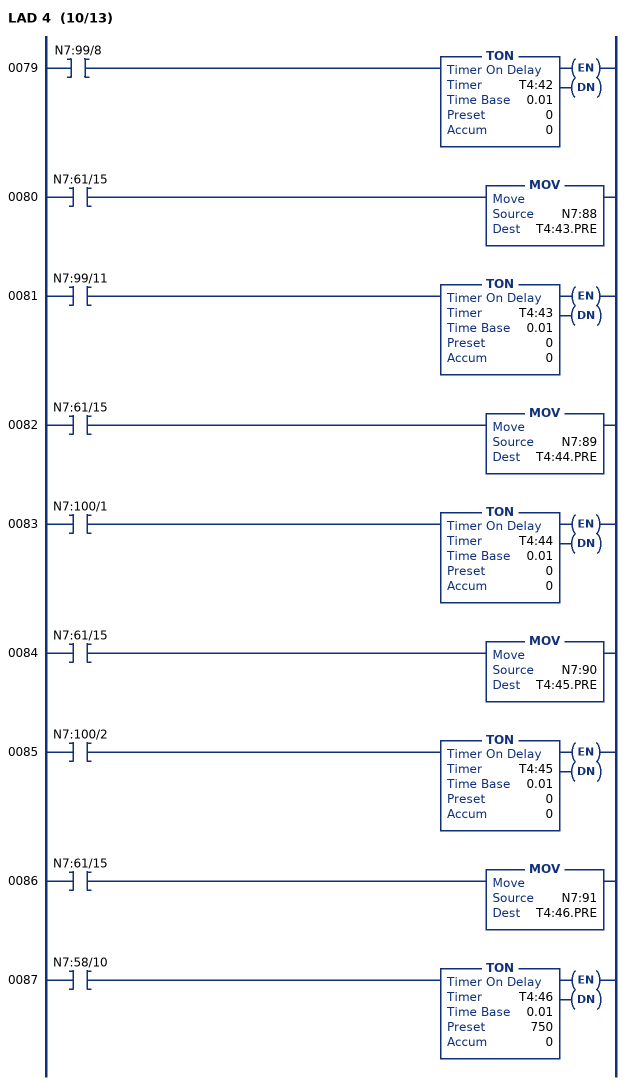
% Rung: 79 %
SOR XIC N7:99/8 TON T4:42 0.01 0 0 EOR
% Rung: 80 %
SOR XIC N7:61/15 MOV N7:88 T4:43.PRE EOR
% Rung: 81 %
SOR XIC N7:99/11 TON T4:43 0.01 0 0 EOR
% Rung: 82 %
SOR XIC N7:61/15 MOV N7:89 T4:44.PRE EOR
% Rung: 83 %
SOR XIC N7:100/1 TON T4:44 0.01 0 0 EOR
% Rung: 84 %
SOR XIC N7:61/15 MOV N7:90 T4:45.PRE EOR
% Rung: 85 %
SOR XIC N7:100/2 TON T4:45 0.01 0 0 EOR
% Rung: 86 %
SOR XIC N7:61/15 MOV N7:91 T4:46.PRE EOR
% Rung: 87 %
SOR XIC N7:58/10 TON T4:46 0.01 750 0 EOR

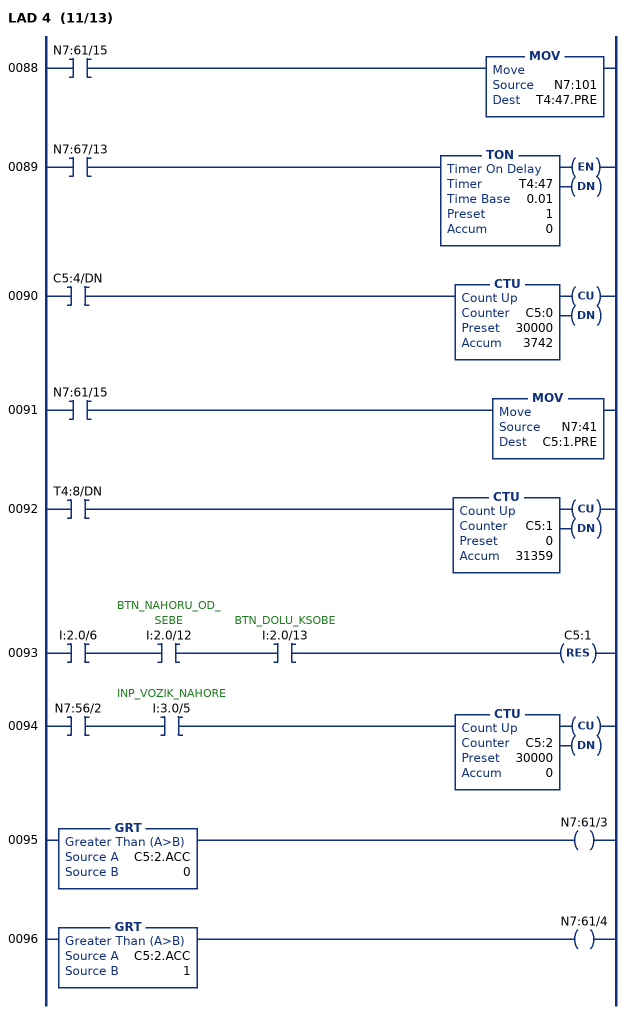
% Rung: 88 %
SOR XIC N7:61/15 MOV N7:101 T4:47.PRE EOR
% Rung: 89 %
SOR XIC N7:67/13 TON T4:47 0.01 1 0 EOR
% Rung: 90 %
SOR XIC C5:4/DN CTU C5:0 30000 3742 EOR
% Rung: 91 %
SOR XIC N7:61/15 MOV N7:41 C5:1.PRE EOR
% Rung: 92 %
SOR XIC T4:8/DN CTU C5:1 0 31359 EOR
% Rung: 93 %
SOR XIC I:2.0/6 XIC I:2.0/12 XIC I:2.0/13 RES C5:1 EOR
%   I:2.0/12  BTN_NAHORU_OD_SEBE %
%   I:2.0/13  BTN_DOLU_KSOBE %
% Rung: 94 %
SOR XIC N7:56/2 XIC I:3.0/5 CTU C5:2 30000 0 EOR
%   I:3.0/5  INP_VOZIK_NAHORE %
% Rung: 95 %
SOR GRT C5:2.ACC 0 OTE N7:61/3 EOR
% Rung: 96 %
SOR GRT C5:2.ACC 1 OTE N7:61/4 EOR

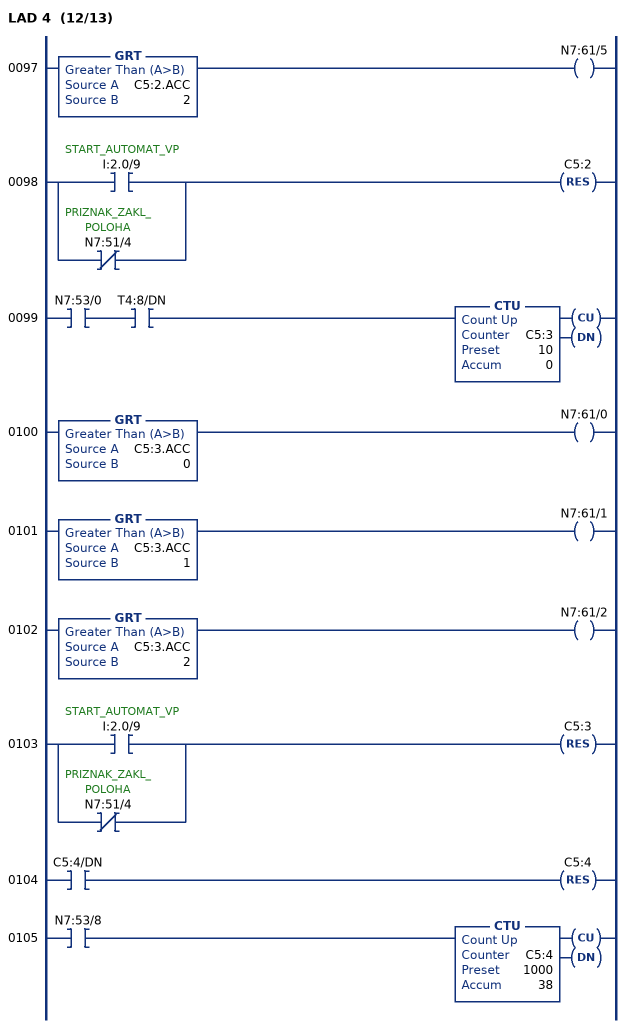
% Rung: 97 %
SOR GRT C5:2.ACC 2 OTE N7:61/5 EOR
% Rung: 98 %
SOR BST XIC I:2.0/9 NXB XIO N7:51/4 BND RES C5:2 EOR
%   I:2.0/9  START_AUTOMAT_VP %
%   N7:51/4  PRIZNAK_ZAKL_POLOHA %
% Rung: 99 %
SOR XIC N7:53/0 XIC T4:8/DN CTU C5:3 10 0 EOR
% Rung: 100 %
SOR GRT C5:3.ACC 0 OTE N7:61/0 EOR
% Rung: 101 %
SOR GRT C5:3.ACC 1 OTE N7:61/1 EOR
% Rung: 102 %
SOR GRT C5:3.ACC 2 OTE N7:61/2 EOR
% Rung: 103 %
SOR BST XIC I:2.0/9 NXB XIO N7:51/4 BND RES C5:3 EOR
%   I:2.0/9  START_AUTOMAT_VP %
%   N7:51/4  PRIZNAK_ZAKL_POLOHA %
% Rung: 104 %
SOR XIC C5:4/DN RES C5:4 EOR
% Rung: 105 %
SOR XIC N7:53/8 CTU C5:4 1000 38 EOR

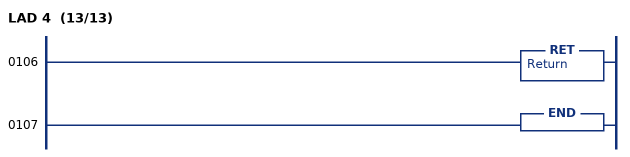
% Rung: 106 %
SOR RET EOR
% Rung: 107 %
SOR END EOR

LADDER 5
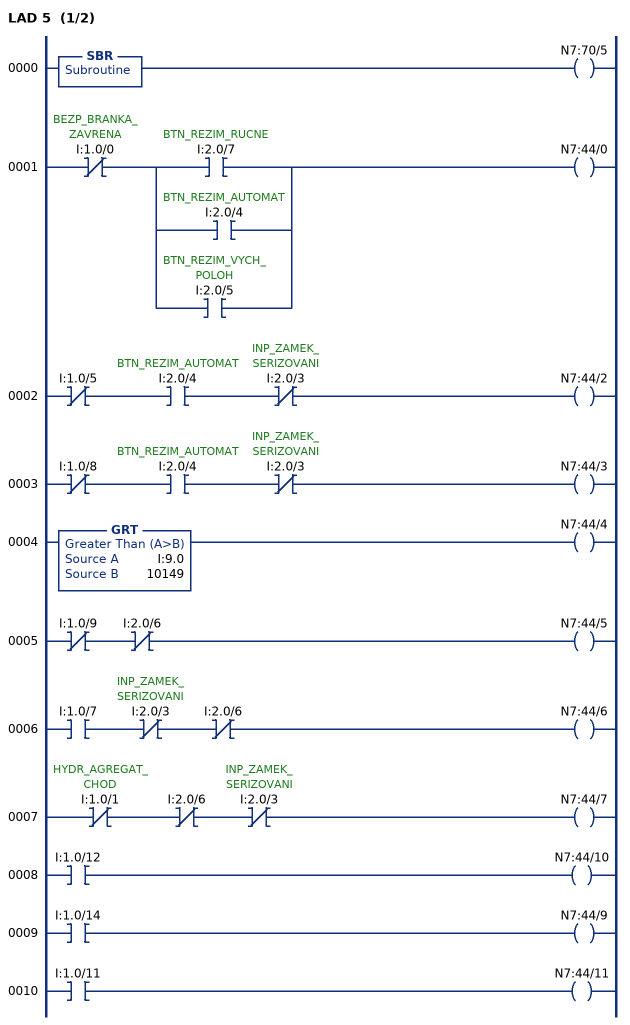
% Rung: 0 %
SOR SBR OTE N7:70/5 EOR
% Rung: 1 %
SOR XIO I:1.0/0 BST XIC I:2.0/7 NXB XIC I:2.0/4 NXB XIC I:2.0/5 BND OTE N7:44/0 EOR
%   I:1.0/0  BEZP_BRANKA_ZAVRENA %
%   I:2.0/7  BTN_REZIM_RUCNE %
%   I:2.0/4  BTN_REZIM_AUTOMAT %
%   I:2.0/5  BTN_REZIM_VYCH_POLOH %
% Rung: 2 %
SOR XIO I:1.0/5 XIC I:2.0/4 XIO I:2.0/3 OTE N7:44/2 EOR
%   I:2.0/4  BTN_REZIM_AUTOMAT %
%   I:2.0/3  INP_ZAMEK_SERIZOVANI %
% Rung: 3 %
SOR XIO I:1.0/8 XIC I:2.0/4 XIO I:2.0/3 OTE N7:44/3 EOR
%   I:2.0/4  BTN_REZIM_AUTOMAT %
%   I:2.0/3  INP_ZAMEK_SERIZOVANI %
% Rung: 4 %
SOR GRT I:9.0 10149 OTE N7:44/4 EOR
% Rung: 5 %
SOR XIO I:1.0/9 XIO I:2.0/6 OTE N7:44/5 EOR
% Rung: 6 %
SOR XIC I:1.0/7 XIO I:2.0/3 XIO I:2.0/6 OTE N7:44/6 EOR
%   I:2.0/3  INP_ZAMEK_SERIZOVANI %
% Rung: 7 %
SOR XIO I:1.0/1 XIO I:2.0/6 XIO I:2.0/3 OTE N7:44/7 EOR
%   I:1.0/1  HYDR_AGREGAT_CHOD %
%   I:2.0/3  INP_ZAMEK_SERIZOVANI %
% Rung: 8 %
SOR XIC I:1.0/12 OTE N7:44/10 EOR
% Rung: 9 %
SOR XIC I:1.0/14 OTE N7:44/9 EOR
% Rung: 10 %
SOR XIC I:1.0/11 OTE N7:44/11 EOR

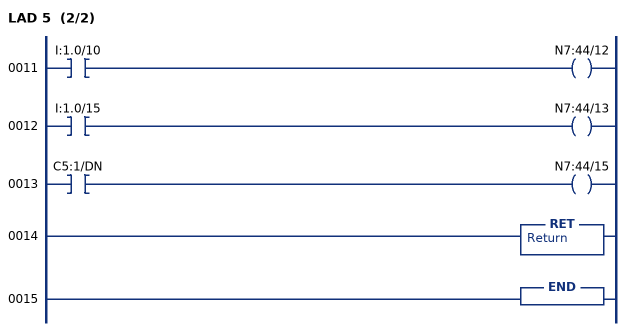
% Rung: 11 %
SOR XIC I:1.0/10 OTE N7:44/12 EOR
% Rung: 12 %
SOR XIC I:1.0/15 OTE N7:44/13 EOR
% Rung: 13 %
SOR XIC C5:1/DN OTE N7:44/15 EOR
% Rung: 14 %
SOR RET EOR
% Rung: 15 %
SOR END EOR

LADDER 6
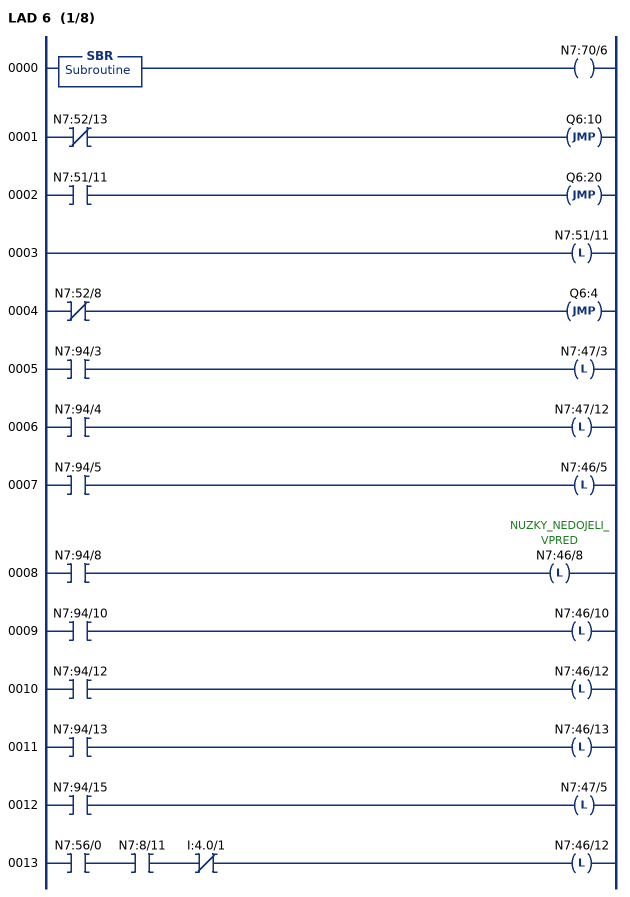
% Rung: 0 %
SOR SBR OTE N7:70/6 EOR
% Rung: 1 %
SOR XIO N7:52/13 JMP Q6:10 EOR
% Rung: 2 %
SOR XIC N7:51/11 JMP Q6:20 EOR
% Rung: 3 %
SOR OTL N7:51/11 EOR
% Rung: 4 %
SOR XIO N7:52/8 JMP Q6:4 EOR
% Rung: 5 %
SOR XIC N7:94/3 OTL N7:47/3 EOR
% Rung: 6 %
SOR XIC N7:94/4 OTL N7:47/12 EOR
% Rung: 7 %
SOR XIC N7:94/5 OTL N7:46/5 EOR
% Rung: 8 %
SOR XIC N7:94/8 OTL N7:46/8 EOR
%   N7:46/8  NUZKY_NEDOJELI_VPRED %
% Rung: 9 %
SOR XIC N7:94/10 OTL N7:46/10 EOR
% Rung: 10 %
SOR XIC N7:94/12 OTL N7:46/12 EOR
% Rung: 11 %
SOR XIC N7:94/13 OTL N7:46/13 EOR
% Rung: 12 %
SOR XIC N7:94/15 OTL N7:47/5 EOR
% Rung: 13 %
SOR XIC N7:56/0 XIC N7:8/11 XIO I:4.0/1 OTL N7:46/12 EOR

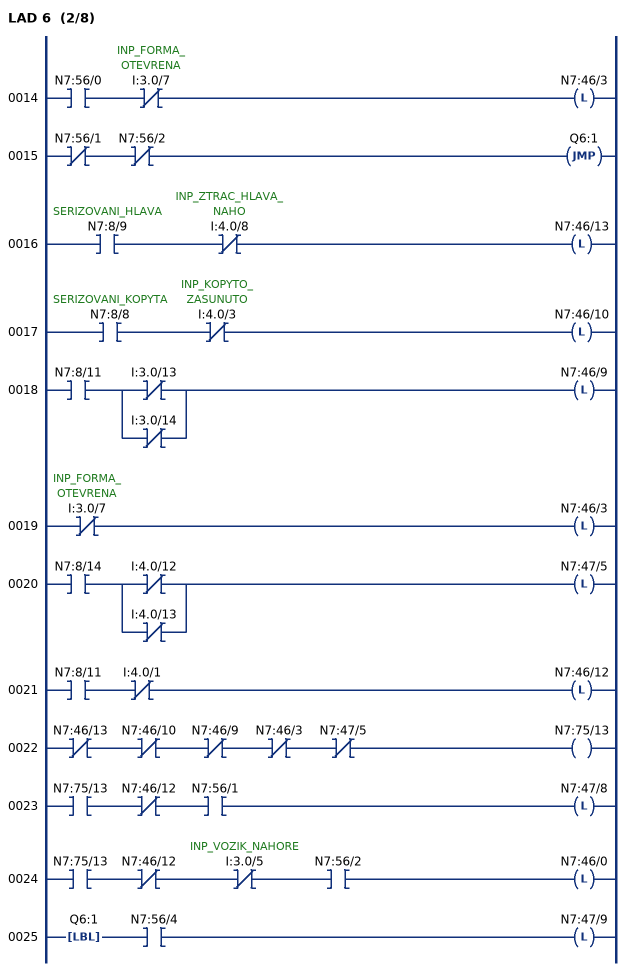
% Rung: 14 %
SOR XIC N7:56/0 XIO I:3.0/7 OTL N7:46/3 EOR
%   I:3.0/7  INP_FORMA_OTEVRENA %
% Rung: 15 %
SOR XIO N7:56/1 XIO N7:56/2 JMP Q6:1 EOR
% Rung: 16 %
SOR XIC N7:8/9 XIO I:4.0/8 OTL N7:46/13 EOR
%   N7:8/9  SERIZOVANI_HLAVA %
%   I:4.0/8  INP_ZTRAC_HLAVA_NAHO %
% Rung: 17 %
SOR XIC N7:8/8 XIO I:4.0/3 OTL N7:46/10 EOR
%   N7:8/8  SERIZOVANI_KOPYTA %
%   I:4.0/3  INP_KOPYTO_ZASUNUTO %
% Rung: 18 %
SOR XIC N7:8/11 BST XIO I:3.0/13 NXB XIO I:3.0/14 BND OTL N7:46/9 EOR
% Rung: 19 %
SOR XIO I:3.0/7 OTL N7:46/3 EOR
%   I:3.0/7  INP_FORMA_OTEVRENA %
% Rung: 20 %
SOR XIC N7:8/14 BST XIO I:4.0/12 NXB XIO I:4.0/13 BND OTL N7:47/5 EOR
% Rung: 21 %
SOR XIC N7:8/11 XIO I:4.0/1 OTL N7:46/12 EOR
% Rung: 22 %
SOR XIO N7:46/13 XIO N7:46/10 XIO N7:46/9 XIO N7:46/3 XIO N7:47/5 OTE N7:75/13 EOR
% Rung: 23 %
SOR XIC N7:75/13 XIO N7:46/12 XIC N7:56/1 OTL N7:47/8 EOR
% Rung: 24 %
SOR XIC N7:75/13 XIO N7:46/12 XIO I:3.0/5 XIC N7:56/2 OTL N7:46/0 EOR
%   I:3.0/5  INP_VOZIK_NAHORE %
% Rung: 25 %
SOR LBL Q6:1 XIC N7:56/4 OTL N7:47/9 EOR

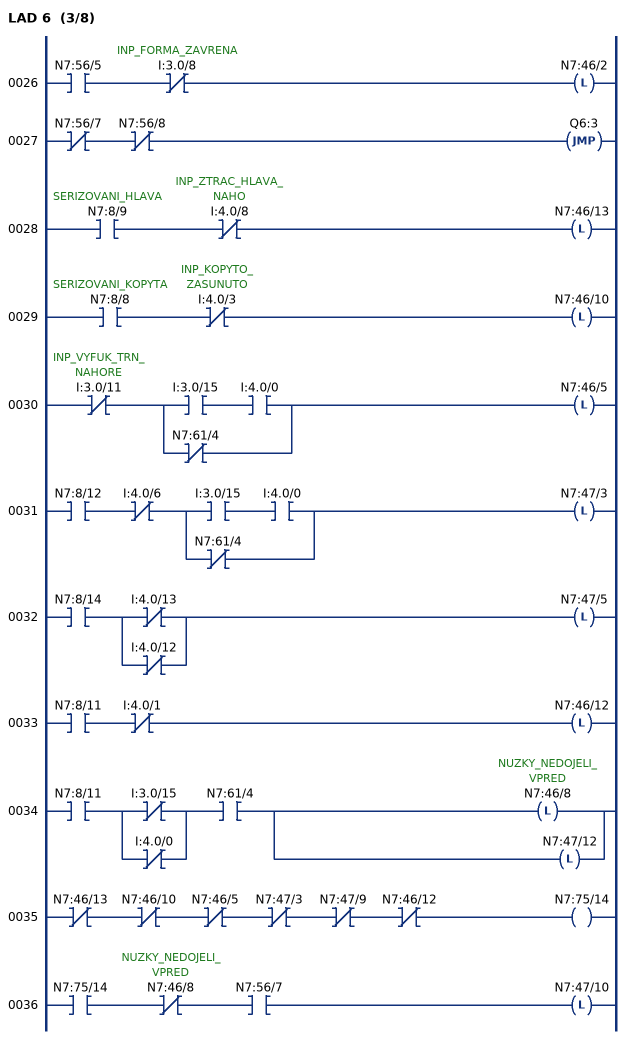
% Rung: 26 %
SOR XIC N7:56/5 XIO I:3.0/8 OTL N7:46/2 EOR
%   I:3.0/8  INP_FORMA_ZAVRENA %
% Rung: 27 %
SOR XIO N7:56/7 XIO N7:56/8 JMP Q6:3 EOR
% Rung: 28 %
SOR XIC N7:8/9 XIO I:4.0/8 OTL N7:46/13 EOR
%   N7:8/9  SERIZOVANI_HLAVA %
%   I:4.0/8  INP_ZTRAC_HLAVA_NAHO %
% Rung: 29 %
SOR XIC N7:8/8 XIO I:4.0/3 OTL N7:46/10 EOR
%   N7:8/8  SERIZOVANI_KOPYTA %
%   I:4.0/3  INP_KOPYTO_ZASUNUTO %
% Rung: 30 %
SOR XIO I:3.0/11 BST XIC I:3.0/15 XIC I:4.0/0 NXB XIO N7:61/4 BND OTL N7:46/5 EOR
%   I:3.0/11  INP_VYFUK_TRN_NAHORE %
% Rung: 31 %
SOR XIC N7:8/12 XIO I:4.0/6 BST XIC I:3.0/15 XIC I:4.0/0 NXB XIO N7:61/4 BND OTL N7:47/3 EOR
% Rung: 32 %
SOR XIC N7:8/14 BST XIO I:4.0/13 NXB XIO I:4.0/12 BND OTL N7:47/5 EOR
% Rung: 33 %
SOR XIC N7:8/11 XIO I:4.0/1 OTL N7:46/12 EOR
% Rung: 34 %
SOR XIC N7:8/11 BST XIO I:3.0/15 NXB XIO I:4.0/0 BND XIC N7:61/4 BST OTL N7:46/8 NXB OTL N7:47/12 BND EOR
%   N7:46/8  NUZKY_NEDOJELI_VPRED %
% Rung: 35 %
SOR XIO N7:46/13 XIO N7:46/10 XIO N7:46/5 XIO N7:47/3 XIO N7:47/9 XIO N7:46/12 OTE N7:75/14 EOR
% Rung: 36 %
SOR XIC N7:75/14 XIO N7:46/8 XIC N7:56/7 OTL N7:47/10 EOR
%   N7:46/8  NUZKY_NEDOJELI_VPRED %

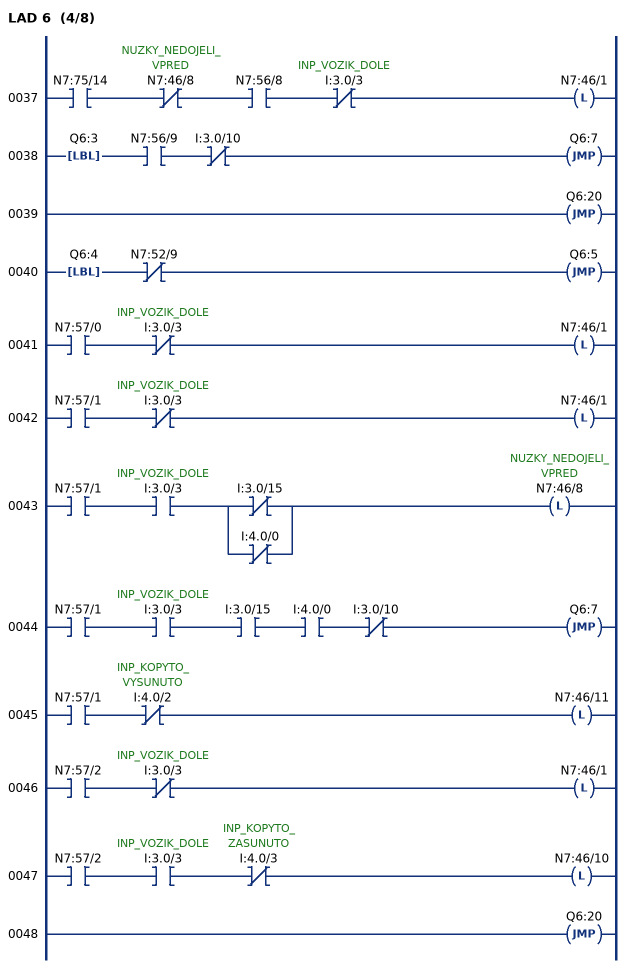
% Rung: 37 %
SOR XIC N7:75/14 XIO N7:46/8 XIC N7:56/8 XIO I:3.0/3 OTL N7:46/1 EOR
%   N7:46/8  NUZKY_NEDOJELI_VPRED %
%   I:3.0/3  INP_VOZIK_DOLE %
% Rung: 38 %
SOR LBL Q6:3 XIC N7:56/9 XIO I:3.0/10 JMP Q6:7 EOR
% Rung: 39 %
SOR JMP Q6:20 EOR
% Rung: 40 %
SOR LBL Q6:4 XIO N7:52/9 JMP Q6:5 EOR
% Rung: 41 %
SOR XIC N7:57/0 XIO I:3.0/3 OTL N7:46/1 EOR
%   I:3.0/3  INP_VOZIK_DOLE %
% Rung: 42 %
SOR XIC N7:57/1 XIO I:3.0/3 OTL N7:46/1 EOR
%   I:3.0/3  INP_VOZIK_DOLE %
% Rung: 43 %
SOR XIC N7:57/1 XIC I:3.0/3 BST XIO I:3.0/15 NXB XIO I:4.0/0 BND OTL N7:46/8 EOR
%   I:3.0/3  INP_VOZIK_DOLE %
%   N7:46/8  NUZKY_NEDOJELI_VPRED %
% Rung: 44 %
SOR XIC N7:57/1 XIC I:3.0/3 XIC I:3.0/15 XIC I:4.0/0 XIO I:3.0/10 JMP Q6:7 EOR
%   I:3.0/3  INP_VOZIK_DOLE %
% Rung: 45 %
SOR XIC N7:57/1 XIO I:4.0/2 OTL N7:46/11 EOR
%   I:4.0/2  INP_KOPYTO_VYSUNUTO %
% Rung: 46 %
SOR XIC N7:57/2 XIO I:3.0/3 OTL N7:46/1 EOR
%   I:3.0/3  INP_VOZIK_DOLE %
% Rung: 47 %
SOR XIC N7:57/2 XIC I:3.0/3 XIO I:4.0/3 OTL N7:46/10 EOR
%   I:3.0/3  INP_VOZIK_DOLE %
%   I:4.0/3  INP_KOPYTO_ZASUNUTO %
% Rung: 48 %
SOR JMP Q6:20 EOR

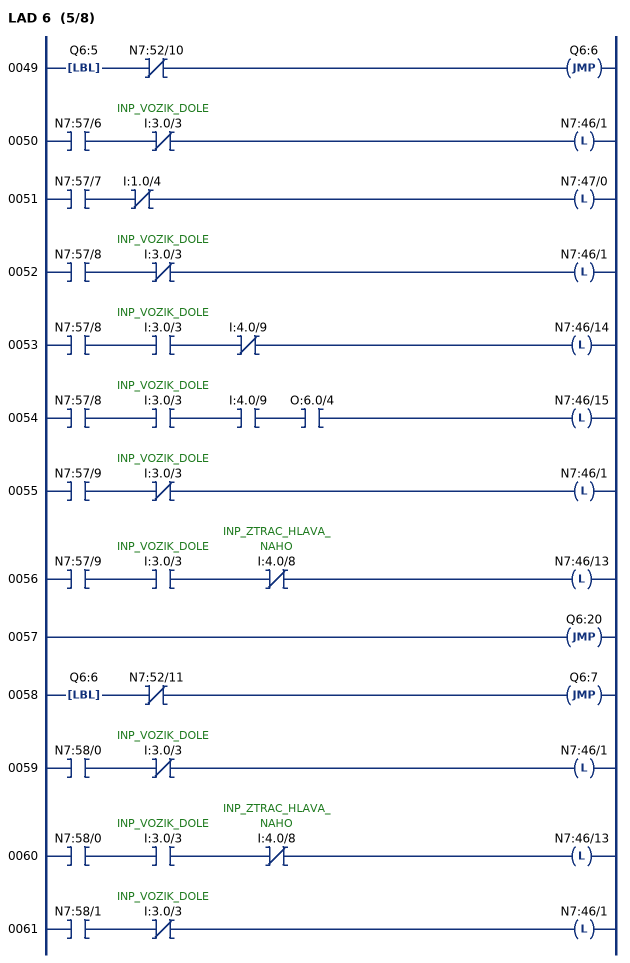
% Rung: 49 %
SOR LBL Q6:5 XIO N7:52/10 JMP Q6:6 EOR
% Rung: 50 %
SOR XIC N7:57/6 XIO I:3.0/3 OTL N7:46/1 EOR
%   I:3.0/3  INP_VOZIK_DOLE %
% Rung: 51 %
SOR XIC N7:57/7 XIO I:1.0/4 OTL N7:47/0 EOR
% Rung: 52 %
SOR XIC N7:57/8 XIO I:3.0/3 OTL N7:46/1 EOR
%   I:3.0/3  INP_VOZIK_DOLE %
% Rung: 53 %
SOR XIC N7:57/8 XIC I:3.0/3 XIO I:4.0/9 OTL N7:46/14 EOR
%   I:3.0/3  INP_VOZIK_DOLE %
% Rung: 54 %
SOR XIC N7:57/8 XIC I:3.0/3 XIC I:4.0/9 XIC O:6.0/4 OTL N7:46/15 EOR
%   I:3.0/3  INP_VOZIK_DOLE %
% Rung: 55 %
SOR XIC N7:57/9 XIO I:3.0/3 OTL N7:46/1 EOR
%   I:3.0/3  INP_VOZIK_DOLE %
% Rung: 56 %
SOR XIC N7:57/9 XIC I:3.0/3 XIO I:4.0/8 OTL N7:46/13 EOR
%   I:3.0/3  INP_VOZIK_DOLE %
%   I:4.0/8  INP_ZTRAC_HLAVA_NAHO %
% Rung: 57 %
SOR JMP Q6:20 EOR
% Rung: 58 %
SOR LBL Q6:6 XIO N7:52/11 JMP Q6:7 EOR
% Rung: 59 %
SOR XIC N7:58/0 XIO I:3.0/3 OTL N7:46/1 EOR
%   I:3.0/3  INP_VOZIK_DOLE %
% Rung: 60 %
SOR XIC N7:58/0 XIC I:3.0/3 XIO I:4.0/8 OTL N7:46/13 EOR
%   I:3.0/3  INP_VOZIK_DOLE %
%   I:4.0/8  INP_ZTRAC_HLAVA_NAHO %
% Rung: 61 %
SOR XIC N7:58/1 XIO I:3.0/3 OTL N7:46/1 EOR
%   I:3.0/3  INP_VOZIK_DOLE %

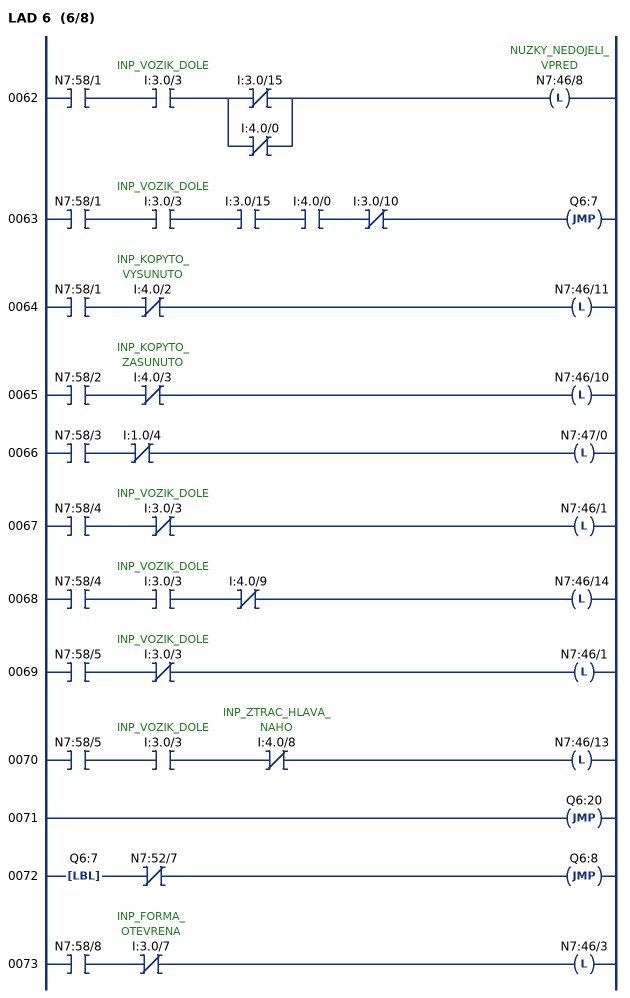
% Rung: 62 %
SOR XIC N7:58/1 XIC I:3.0/3 BST XIO I:3.0/15 NXB XIO I:4.0/0 BND OTL N7:46/8 EOR
%   I:3.0/3  INP_VOZIK_DOLE %
%   N7:46/8  NUZKY_NEDOJELI_VPRED %
% Rung: 63 %
SOR XIC N7:58/1 XIC I:3.0/3 XIC I:3.0/15 XIC I:4.0/0 XIO I:3.0/10 JMP Q6:7 EOR
%   I:3.0/3  INP_VOZIK_DOLE %
% Rung: 64 %
SOR XIC N7:58/1 XIO I:4.0/2 OTL N7:46/11 EOR
%   I:4.0/2  INP_KOPYTO_VYSUNUTO %
% Rung: 65 %
SOR XIC N7:58/2 XIO I:4.0/3 OTL N7:46/10 EOR
%   I:4.0/3  INP_KOPYTO_ZASUNUTO %
% Rung: 66 %
SOR XIC N7:58/3 XIO I:1.0/4 OTL N7:47/0 EOR
% Rung: 67 %
SOR XIC N7:58/4 XIO I:3.0/3 OTL N7:46/1 EOR
%   I:3.0/3  INP_VOZIK_DOLE %
% Rung: 68 %
SOR XIC N7:58/4 XIC I:3.0/3 XIO I:4.0/9 OTL N7:46/14 EOR
%   I:3.0/3  INP_VOZIK_DOLE %
% Rung: 69 %
SOR XIC N7:58/5 XIO I:3.0/3 OTL N7:46/1 EOR
%   I:3.0/3  INP_VOZIK_DOLE %
% Rung: 70 %
SOR XIC N7:58/5 XIC I:3.0/3 XIO I:4.0/8 OTL N7:46/13 EOR
%   I:3.0/3  INP_VOZIK_DOLE %
%   I:4.0/8  INP_ZTRAC_HLAVA_NAHO %
% Rung: 71 %
SOR JMP Q6:20 EOR
% Rung: 72 %
SOR LBL Q6:7 XIO N7:52/7 JMP Q6:8 EOR
% Rung: 73 %
SOR XIC N7:58/8 XIO I:3.0/7 OTL N7:46/3 EOR
%   I:3.0/7  INP_FORMA_OTEVRENA %

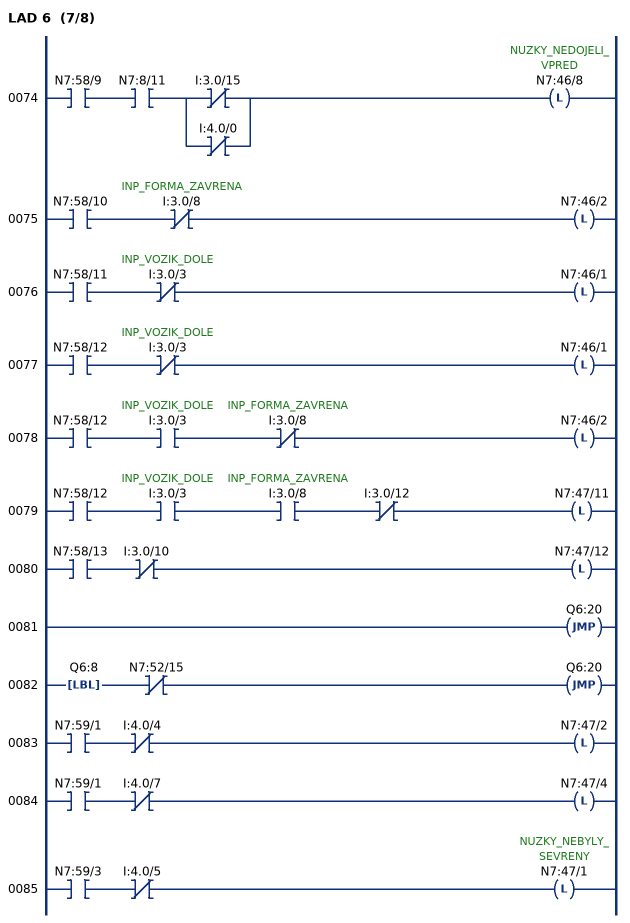
% Rung: 74 %
SOR XIC N7:58/9 XIC N7:8/11 BST XIO I:3.0/15 NXB XIO I:4.0/0 BND OTL N7:46/8 EOR
%   N7:46/8  NUZKY_NEDOJELI_VPRED %
% Rung: 75 %
SOR XIC N7:58/10 XIO I:3.0/8 OTL N7:46/2 EOR
%   I:3.0/8  INP_FORMA_ZAVRENA %
% Rung: 76 %
SOR XIC N7:58/11 XIO I:3.0/3 OTL N7:46/1 EOR
%   I:3.0/3  INP_VOZIK_DOLE %
% Rung: 77 %
SOR XIC N7:58/12 XIO I:3.0/3 OTL N7:46/1 EOR
%   I:3.0/3  INP_VOZIK_DOLE %
% Rung: 78 %
SOR XIC N7:58/12 XIC I:3.0/3 XIO I:3.0/8 OTL N7:46/2 EOR
%   I:3.0/3  INP_VOZIK_DOLE %
%   I:3.0/8  INP_FORMA_ZAVRENA %
% Rung: 79 %
SOR XIC N7:58/12 XIC I:3.0/3 XIC I:3.0/8 XIO I:3.0/12 OTL N7:47/11 EOR
%   I:3.0/3  INP_VOZIK_DOLE %
%   I:3.0/8  INP_FORMA_ZAVRENA %
% Rung: 80 %
SOR XIC N7:58/13 XIO I:3.0/10 OTL N7:47/12 EOR
% Rung: 81 %
SOR JMP Q6:20 EOR
% Rung: 82 %
SOR LBL Q6:8 XIO N7:52/15 JMP Q6:20 EOR
% Rung: 83 %
SOR XIC N7:59/1 XIO I:4.0/4 OTL N7:47/2 EOR
% Rung: 84 %
SOR XIC N7:59/1 XIO I:4.0/7 OTL N7:47/4 EOR
% Rung: 85 %
SOR XIC N7:59/3 XIO I:4.0/5 OTL N7:47/1 EOR
%   N7:47/1  NUZKY_NEBYLY_SEVRENY %

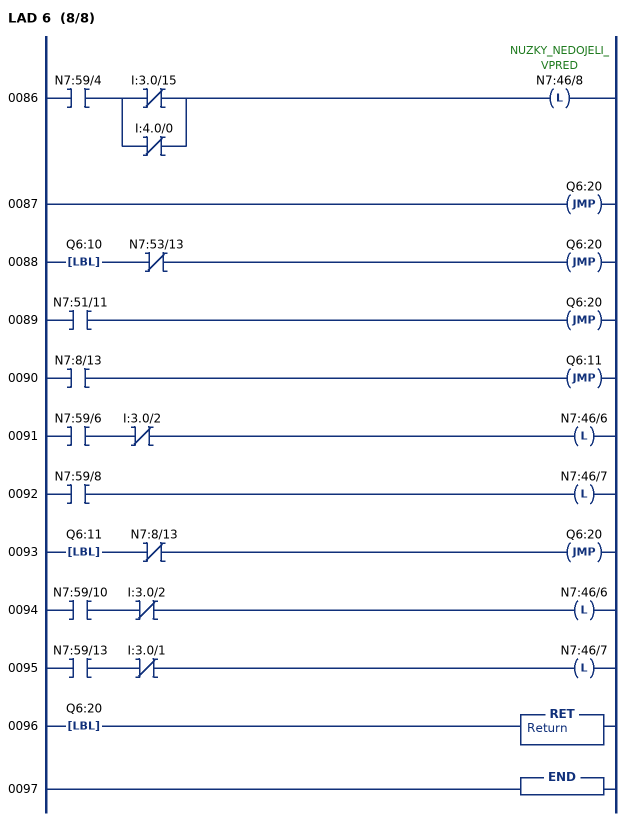
% Rung: 86 %
SOR XIC N7:59/4 BST XIO I:3.0/15 NXB XIO I:4.0/0 BND OTL N7:46/8 EOR
%   N7:46/8  NUZKY_NEDOJELI_VPRED %
% Rung: 87 %
SOR JMP Q6:20 EOR
% Rung: 88 %
SOR LBL Q6:10 XIO N7:53/13 JMP Q6:20 EOR
% Rung: 89 %
SOR XIC N7:51/11 JMP Q6:20 EOR
% Rung: 90 %
SOR XIC N7:8/13 JMP Q6:11 EOR
% Rung: 91 %
SOR XIC N7:59/6 XIO I:3.0/2 OTL N7:46/6 EOR
% Rung: 92 %
SOR XIC N7:59/8 OTL N7:46/7 EOR
% Rung: 93 %
SOR LBL Q6:11 XIO N7:8/13 JMP Q6:20 EOR
% Rung: 94 %
SOR XIC N7:59/10 XIO I:3.0/2 OTL N7:46/6 EOR
% Rung: 95 %
SOR XIC N7:59/13 XIO I:3.0/1 OTL N7:46/7 EOR
% Rung: 96 %
SOR LBL Q6:20 RET EOR
% Rung: 97 %
SOR END EOR

LADDER 7
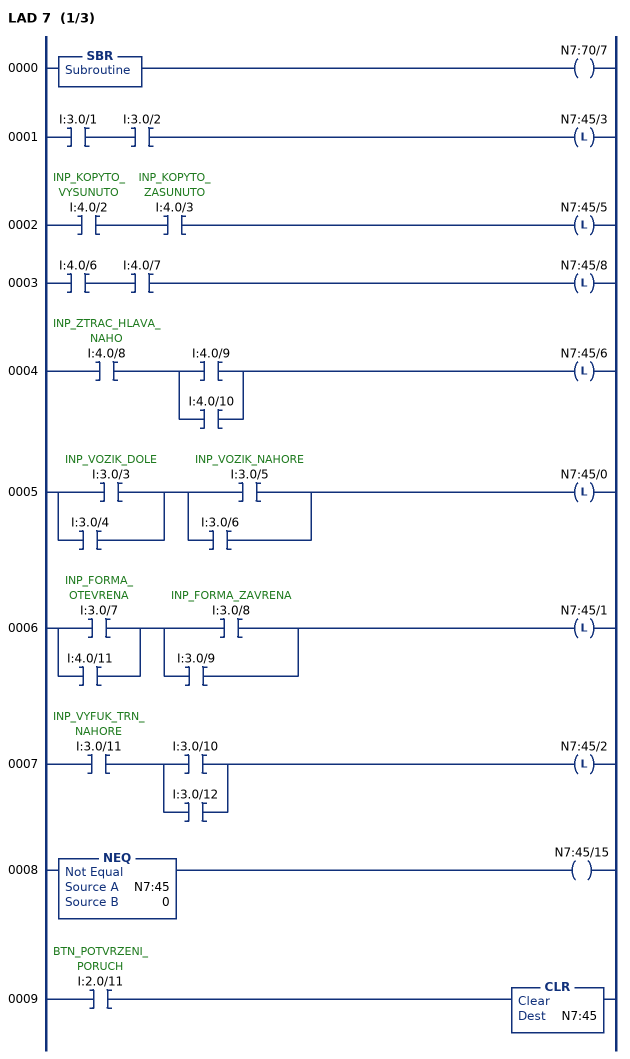
% Rung: 0 %
SOR SBR OTE N7:70/7 EOR
% Rung: 1 %
SOR XIC I:3.0/1 XIC I:3.0/2 OTL N7:45/3 EOR
% Rung: 2 %
SOR XIC I:4.0/2 XIC I:4.0/3 OTL N7:45/5 EOR
%   I:4.0/2  INP_KOPYTO_VYSUNUTO %
%   I:4.0/3  INP_KOPYTO_ZASUNUTO %
% Rung: 3 %
SOR XIC I:4.0/6 XIC I:4.0/7 OTL N7:45/8 EOR
% Rung: 4 %
SOR XIC I:4.0/8 BST XIC I:4.0/9 NXB XIC I:4.0/10 BND OTL N7:45/6 EOR
%   I:4.0/8  INP_ZTRAC_HLAVA_NAHO %
% Rung: 5 %
SOR BST XIC I:3.0/3 NXB XIC I:3.0/4 BND BST XIC I:3.0/5 NXB XIC I:3.0/6 BND OTL N7:45/0 EOR
%   I:3.0/3  INP_VOZIK_DOLE %
%   I:3.0/5  INP_VOZIK_NAHORE %
% Rung: 6 %
SOR BST XIC I:3.0/7 NXB XIC I:4.0/11 BND BST XIC I:3.0/8 NXB XIC I:3.0/9 BND OTL N7:45/1 EOR
%   I:3.0/7  INP_FORMA_OTEVRENA %
%   I:3.0/8  INP_FORMA_ZAVRENA %
% Rung: 7 %
SOR XIC I:3.0/11 BST XIC I:3.0/10 NXB XIC I:3.0/12 BND OTL N7:45/2 EOR
%   I:3.0/11  INP_VYFUK_TRN_NAHORE %
% Rung: 8 %
SOR NEQ N7:45 0 OTE N7:45/15 EOR
% Rung: 9 %
SOR XIC I:2.0/11 CLR N7:45 EOR
%   I:2.0/11  BTN_POTVRZENI_PORUCH %

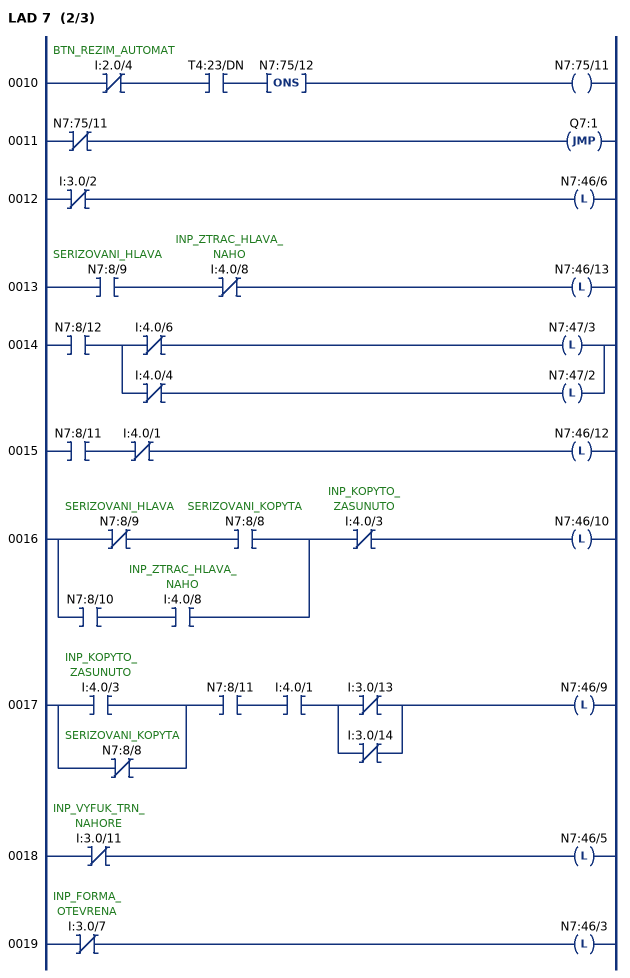
% Rung: 10 %
SOR XIO I:2.0/4 XIC T4:23/DN OSR N7:75/12 OTE N7:75/11 EOR
%   I:2.0/4  BTN_REZIM_AUTOMAT %
% Rung: 11 %
SOR XIO N7:75/11 JMP Q7:1 EOR
% Rung: 12 %
SOR XIO I:3.0/2 OTL N7:46/6 EOR
% Rung: 13 %
SOR XIC N7:8/9 XIO I:4.0/8 OTL N7:46/13 EOR
%   N7:8/9  SERIZOVANI_HLAVA %
%   I:4.0/8  INP_ZTRAC_HLAVA_NAHO %
% Rung: 14 %
SOR XIC N7:8/12 BST XIO I:4.0/6 OTL N7:47/3 NXB XIO I:4.0/4 OTL N7:47/2 BND EOR
% Rung: 15 %
SOR XIC N7:8/11 XIO I:4.0/1 OTL N7:46/12 EOR
% Rung: 16 %
SOR BST XIO N7:8/9 XIC N7:8/8 NXB XIC N7:8/10 XIC I:4.0/8 BND XIO I:4.0/3 OTL N7:46/10 EOR
%   N7:8/9  SERIZOVANI_HLAVA %
%   N7:8/8  SERIZOVANI_KOPYTA %
%   I:4.0/8  INP_ZTRAC_HLAVA_NAHO %
%   I:4.0/3  INP_KOPYTO_ZASUNUTO %
% Rung: 17 %
SOR BST XIC I:4.0/3 NXB XIO N7:8/8 BND XIC N7:8/11 XIC I:4.0/1 BST XIO I:3.0/13 NXB XIO I:3.0/14 BND OTL N7:46/9 EOR
%   I:4.0/3  INP_KOPYTO_ZASUNUTO %
%   N7:8/8  SERIZOVANI_KOPYTA %
% Rung: 18 %
SOR XIO I:3.0/11 OTL N7:46/5 EOR
%   I:3.0/11  INP_VYFUK_TRN_NAHORE %
% Rung: 19 %
SOR XIO I:3.0/7 OTL N7:46/3 EOR
%   I:3.0/7  INP_FORMA_OTEVRENA %

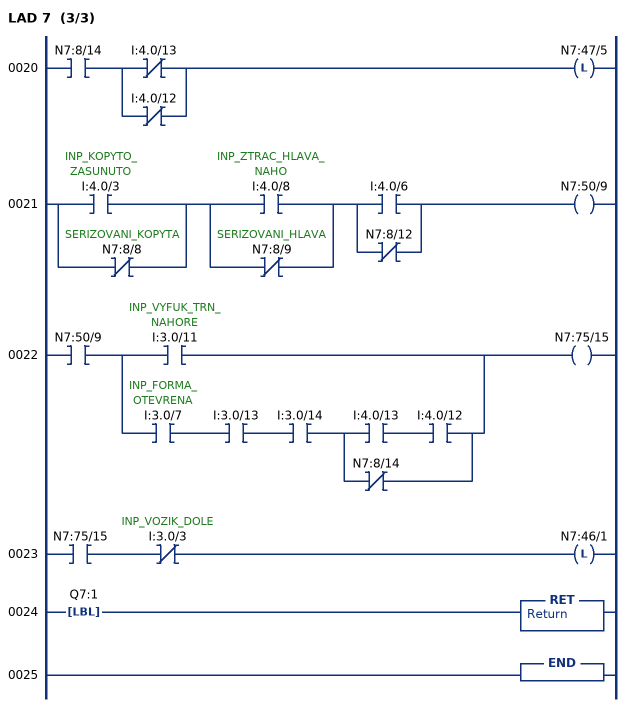
% Rung: 20 %
SOR XIC N7:8/14 BST XIO I:4.0/13 NXB XIO I:4.0/12 BND OTL N7:47/5 EOR
% Rung: 21 %
SOR BST XIC I:4.0/3 NXB XIO N7:8/8 BND BST XIC I:4.0/8 NXB XIO N7:8/9 BND BST XIC I:4.0/6 NXB XIO N7:8/12 BND OTE N7:50/9 EOR
%   I:4.0/3  INP_KOPYTO_ZASUNUTO %
%   N7:8/8  SERIZOVANI_KOPYTA %
%   I:4.0/8  INP_ZTRAC_HLAVA_NAHO %
%   N7:8/9  SERIZOVANI_HLAVA %
% Rung: 22 %
SOR XIC N7:50/9 BST XIC I:3.0/11 NXB XIC I:3.0/7 XIC I:3.0/13 XIC I:3.0/14 BST XIC I:4.0/13 XIC I:4.0/12 NXB XIO N7:8/14 BND BND OTE N7:75/15 EOR
%   I:3.0/11  INP_VYFUK_TRN_NAHORE %
%   I:3.0/7  INP_FORMA_OTEVRENA %
% Rung: 23 %
SOR XIC N7:75/15 XIO I:3.0/3 OTL N7:46/1 EOR
%   I:3.0/3  INP_VOZIK_DOLE %
% Rung: 24 %
SOR LBL Q7:1 RET EOR
% Rung: 25 %
SOR END EOR

LADDER 8
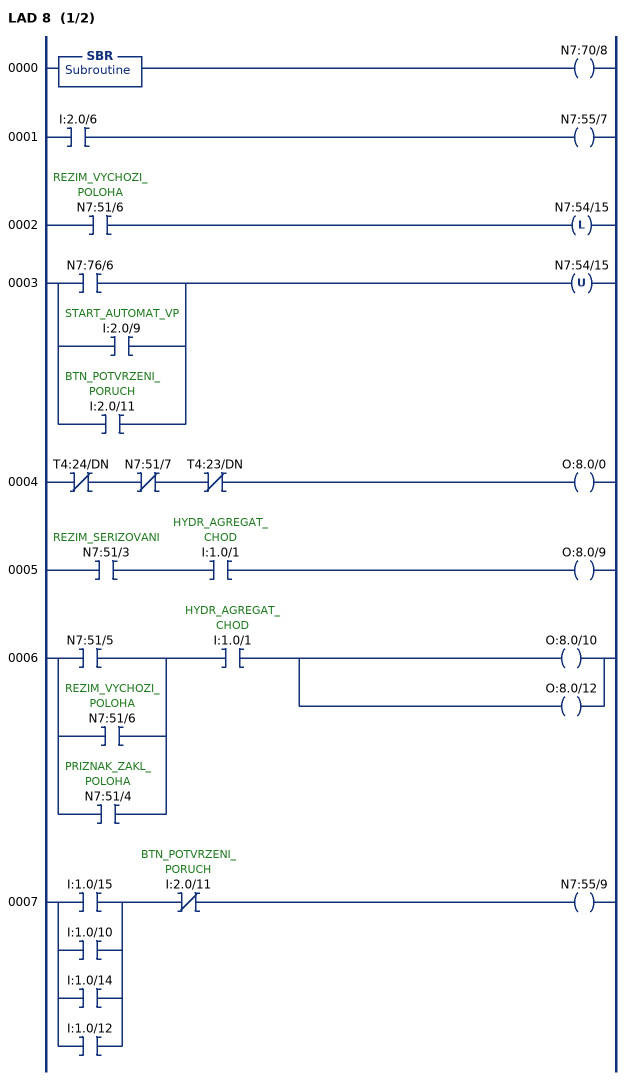
% Rung: 0 %
SOR SBR OTE N7:70/8 EOR
% Rung: 1 %
SOR XIC I:2.0/6 OTE N7:55/7 EOR
% Rung: 2 %
SOR XIC N7:51/6 OTL N7:54/15 EOR
%   N7:51/6  REZIM_VYCHOZI_POLOHA %
% Rung: 3 %
SOR BST XIC N7:76/6 NXB XIC I:2.0/9 NXB XIC I:2.0/11 BND OTU N7:54/15 EOR
%   I:2.0/9  START_AUTOMAT_VP %
%   I:2.0/11  BTN_POTVRZENI_PORUCH %
% Rung: 4 %
SOR XIO T4:24/DN XIO N7:51/7 XIO T4:23/DN OTE O:8.0/0 EOR
% Rung: 5 %
SOR XIC N7:51/3 XIC I:1.0/1 OTE O:8.0/9 EOR
%   N7:51/3  REZIM_SERIZOVANI %
%   I:1.0/1  HYDR_AGREGAT_CHOD %
% Rung: 6 %
SOR BST XIC N7:51/5 NXB XIC N7:51/6 NXB XIC N7:51/4 BND XIC I:1.0/1 BST OTE O:8.0/10 NXB OTE O:8.0/12 BND EOR
%   N7:51/6  REZIM_VYCHOZI_POLOHA %
%   N7:51/4  PRIZNAK_ZAKL_POLOHA %
%   I:1.0/1  HYDR_AGREGAT_CHOD %
% Rung: 7 %
SOR BST XIC I:1.0/15 NXB XIC I:1.0/10 NXB XIC I:1.0/14 NXB XIC I:1.0/12 BND XIO I:2.0/11 OTE N7:55/9 EOR
%   I:2.0/11  BTN_POTVRZENI_PORUCH %

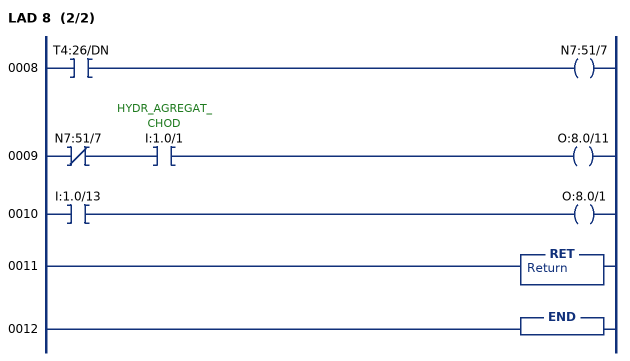
% Rung: 8 %
SOR XIC T4:26/DN OTE N7:51/7 EOR
% Rung: 9 %
SOR XIO N7:51/7 XIC I:1.0/1 OTE O:8.0/11 EOR
%   I:1.0/1  HYDR_AGREGAT_CHOD %
% Rung: 10 %
SOR XIC I:1.0/13 OTE O:8.0/1 EOR
% Rung: 11 %
SOR RET EOR
% Rung: 12 %
SOR END EOR

LADDER 9
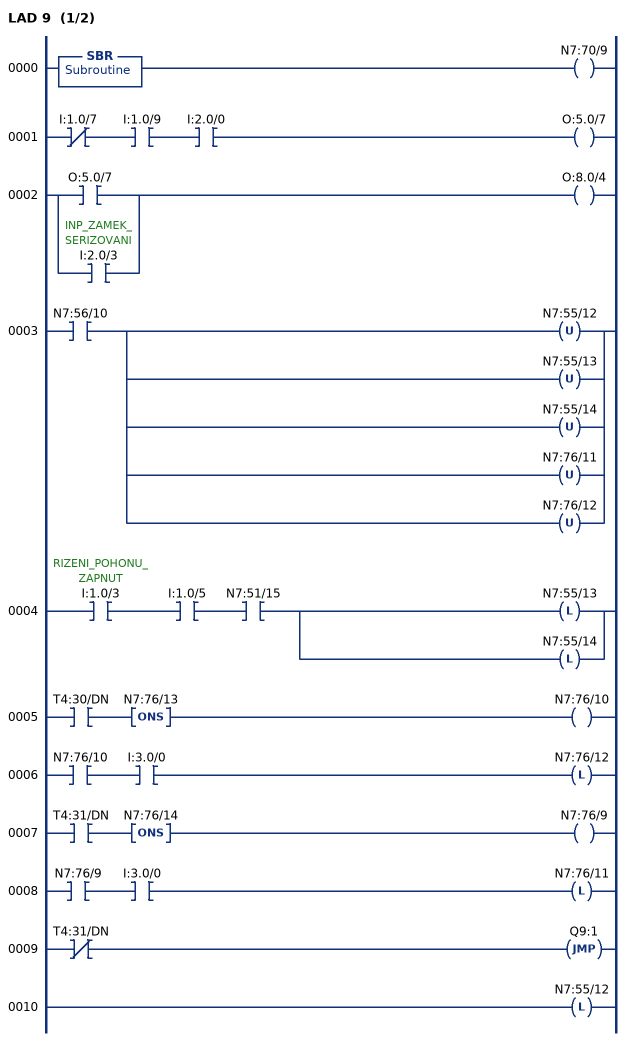
% Rung: 0 %
SOR SBR OTE N7:70/9 EOR
% Rung: 1 %
SOR XIO I:1.0/7 XIC I:1.0/9 XIC I:2.0/0 OTE O:5.0/7 EOR
% Rung: 2 %
SOR BST XIC O:5.0/7 NXB XIC I:2.0/3 BND OTE O:8.0/4 EOR
%   I:2.0/3  INP_ZAMEK_SERIZOVANI %
% Rung: 3 %
SOR XIC N7:56/10 BST OTU N7:55/12 NXB OTU N7:55/13 NXB OTU N7:55/14 NXB OTU N7:76/11 NXB OTU N7:76/12 BND EOR
% Rung: 4 %
SOR XIC I:1.0/3 XIC I:1.0/5 XIC N7:51/15 BST OTL N7:55/13 NXB OTL N7:55/14 BND EOR
%   I:1.0/3  RIZENI_POHONU_ZAPNUT %
% Rung: 5 %
SOR XIC T4:30/DN OSR N7:76/13 OTE N7:76/10 EOR
% Rung: 6 %
SOR XIC N7:76/10 XIC I:3.0/0 OTL N7:76/12 EOR
% Rung: 7 %
SOR XIC T4:31/DN OSR N7:76/14 OTE N7:76/9 EOR
% Rung: 8 %
SOR XIC N7:76/9 XIC I:3.0/0 OTL N7:76/11 EOR
% Rung: 9 %
SOR XIO T4:31/DN JMP Q9:1 EOR
% Rung: 10 %
SOR OTL N7:55/12 EOR

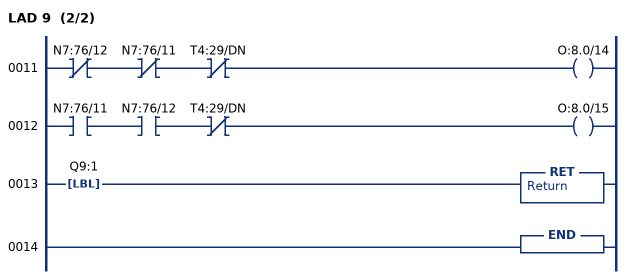
% Rung: 11 %
SOR XIO N7:76/12 XIO N7:76/11 XIO T4:29/DN OTE O:8.0/14 EOR
% Rung: 12 %
SOR XIC N7:76/11 XIC N7:76/12 XIO T4:29/DN OTE O:8.0/15 EOR
% Rung: 13 %
SOR LBL Q9:1 RET EOR
% Rung: 14 %
SOR END EOR

LADDER 10
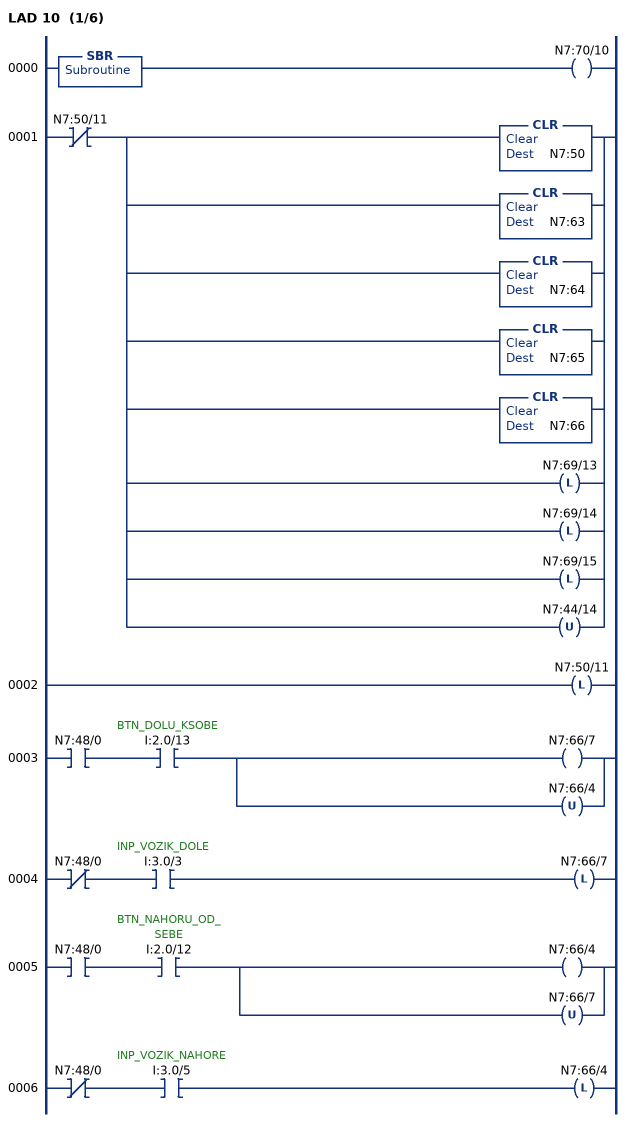
% Rung: 0 %
SOR SBR OTE N7:70/10 EOR
% Rung: 1 %
SOR XIO N7:50/11 BST CLR N7:50 NXB CLR N7:63 NXB CLR N7:64 NXB CLR N7:65 NXB CLR N7:66 NXB OTL N7:69/13 NXB OTL N7:69/14 NXB OTL N7:69/15 NXB OTU N7:44/14 BND EOR
% Rung: 2 %
SOR OTL N7:50/11 EOR
% Rung: 3 %
SOR XIC N7:48/0 XIC I:2.0/13 BST OTE N7:66/7 NXB OTU N7:66/4 BND EOR
%   I:2.0/13  BTN_DOLU_KSOBE %
% Rung: 4 %
SOR XIO N7:48/0 XIC I:3.0/3 OTL N7:66/7 EOR
%   I:3.0/3  INP_VOZIK_DOLE %
% Rung: 5 %
SOR XIC N7:48/0 XIC I:2.0/12 BST OTE N7:66/4 NXB OTU N7:66/7 BND EOR
%   I:2.0/12  BTN_NAHORU_OD_SEBE %
% Rung: 6 %
SOR XIO N7:48/0 XIC I:3.0/5 OTL N7:66/4 EOR
%   I:3.0/5  INP_VOZIK_NAHORE %

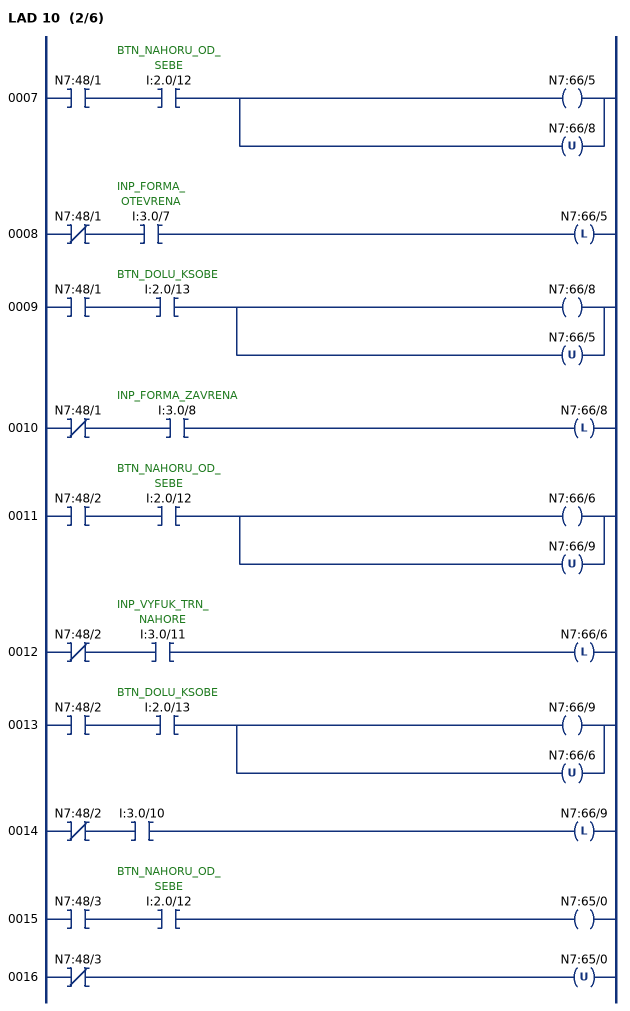
% Rung: 7 %
SOR XIC N7:48/1 XIC I:2.0/12 BST OTE N7:66/5 NXB OTU N7:66/8 BND EOR
%   I:2.0/12  BTN_NAHORU_OD_SEBE %
% Rung: 8 %
SOR XIO N7:48/1 XIC I:3.0/7 OTL N7:66/5 EOR
%   I:3.0/7  INP_FORMA_OTEVRENA %
% Rung: 9 %
SOR XIC N7:48/1 XIC I:2.0/13 BST OTE N7:66/8 NXB OTU N7:66/5 BND EOR
%   I:2.0/13  BTN_DOLU_KSOBE %
% Rung: 10 %
SOR XIO N7:48/1 XIC I:3.0/8 OTL N7:66/8 EOR
%   I:3.0/8  INP_FORMA_ZAVRENA %
% Rung: 11 %
SOR XIC N7:48/2 XIC I:2.0/12 BST OTE N7:66/6 NXB OTU N7:66/9 BND EOR
%   I:2.0/12  BTN_NAHORU_OD_SEBE %
% Rung: 12 %
SOR XIO N7:48/2 XIC I:3.0/11 OTL N7:66/6 EOR
%   I:3.0/11  INP_VYFUK_TRN_NAHORE %
% Rung: 13 %
SOR XIC N7:48/2 XIC I:2.0/13 BST OTE N7:66/9 NXB OTU N7:66/6 BND EOR
%   I:2.0/13  BTN_DOLU_KSOBE %
% Rung: 14 %
SOR XIO N7:48/2 XIC I:3.0/10 OTL N7:66/9 EOR
% Rung: 15 %
SOR XIC N7:48/3 XIC I:2.0/12 OTE N7:65/0 EOR
%   I:2.0/12  BTN_NAHORU_OD_SEBE %
% Rung: 16 %
SOR XIO N7:48/3 OTU N7:65/0 EOR

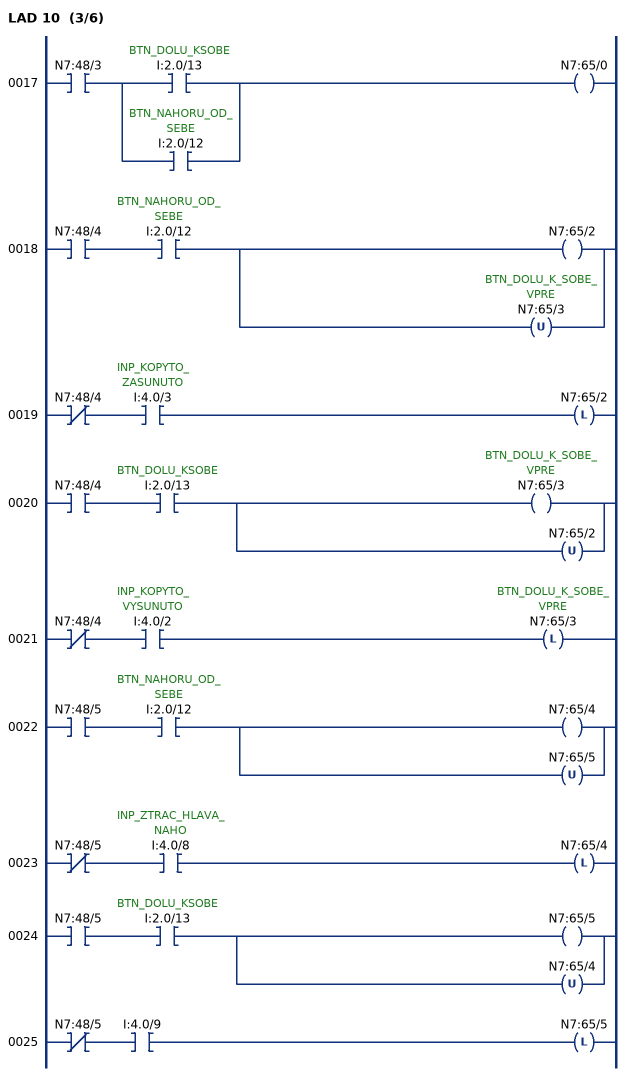
% Rung: 17 %
SOR XIC N7:48/3 BST XIC I:2.0/13 NXB XIC I:2.0/12 BND OTE N7:65/0 EOR
%   I:2.0/13  BTN_DOLU_KSOBE %
%   I:2.0/12  BTN_NAHORU_OD_SEBE %
% Rung: 18 %
SOR XIC N7:48/4 XIC I:2.0/12 BST OTE N7:65/2 NXB OTU N7:65/3 BND EOR
%   I:2.0/12  BTN_NAHORU_OD_SEBE %
%   N7:65/3  BTN_DOLU_K_SOBE_VPRE %
% Rung: 19 %
SOR XIO N7:48/4 XIC I:4.0/3 OTL N7:65/2 EOR
%   I:4.0/3  INP_KOPYTO_ZASUNUTO %
% Rung: 20 %
SOR XIC N7:48/4 XIC I:2.0/13 BST OTE N7:65/3 NXB OTU N7:65/2 BND EOR
%   I:2.0/13  BTN_DOLU_KSOBE %
%   N7:65/3  BTN_DOLU_K_SOBE_VPRE %
% Rung: 21 %
SOR XIO N7:48/4 XIC I:4.0/2 OTL N7:65/3 EOR
%   I:4.0/2  INP_KOPYTO_VYSUNUTO %
%   N7:65/3  BTN_DOLU_K_SOBE_VPRE %
% Rung: 22 %
SOR XIC N7:48/5 XIC I:2.0/12 BST OTE N7:65/4 NXB OTU N7:65/5 BND EOR
%   I:2.0/12  BTN_NAHORU_OD_SEBE %
% Rung: 23 %
SOR XIO N7:48/5 XIC I:4.0/8 OTL N7:65/4 EOR
%   I:4.0/8  INP_ZTRAC_HLAVA_NAHO %
% Rung: 24 %
SOR XIC N7:48/5 XIC I:2.0/13 BST OTE N7:65/5 NXB OTU N7:65/4 BND EOR
%   I:2.0/13  BTN_DOLU_KSOBE %
% Rung: 25 %
SOR XIO N7:48/5 XIC I:4.0/9 OTL N7:65/5 EOR

